{attribute 'pack_mode' := '1'}
TYPE PDFReportResponseStructure :
STRUCT
	ResponseCode : UDINT;
END_STRUCT
END_TYPE

(* stored: Version 1.1.0.1, ProductVersion 3.1.4024.12
   DUT PDFReportResponseStructure: Id {7633e98b-94f8-4a28-8b95-d849fcff87f7} *)
